// TIA Portal V19 export
FUNCTION_BLOCK "TYPIC_C501_SF_DME"   // FB55, FBD
TITLE = TYPIC_C501_SF_DME: Drukmeting
{ S7_Optimized_Access := 'TRUE' }
AUTHOR : OCOTECH
FAMILY : Typical
NAME : C501.813
// Logisch Object Besturing: C501.813
// 
// Het doel van deze subfunctie is om de algemene sturing en bediening vanuit 3B te voorzien van een drukmeting behorende tot de brandblusinstallatie.
// stored: MemoryReserve 10, SetENOAutomatically false
   VAR_INPUT
      CFG_SIG_HH { ExternalAccessible := 'False'; ExternalVisible := 'False'; ExternalWritable := 'False'} : Real;   // Schakeldrempel signalering te hoog
      CFG_SIG_H { ExternalAccessible := 'False'; ExternalVisible := 'False'; ExternalWritable := 'False'} : Real;   // Schakeldrempel signalering voorwaarschuwing hoog
      CFG_HYS_H { ExternalAccessible := 'False'; ExternalVisible := 'False'; ExternalWritable := 'False'} : Real;   // Hysteresis op signalering te hoog en voorwaarschuwing hoog
      CFG_ITYD_H { ExternalAccessible := 'False'; ExternalVisible := 'False'; ExternalWritable := 'False'} : Real;   // Tijdsvertraging signalering te hoog
      CFG_SIG_L { ExternalAccessible := 'False'; ExternalVisible := 'False'; ExternalWritable := 'False'} : Real;   // Schakeldrempel signalering te laag
      CFG_HYS_L { ExternalAccessible := 'False'; ExternalVisible := 'False'; ExternalWritable := 'False'} : Real;   // Hysteresis op signalering te laag
      CFG_ITYD_L { ExternalAccessible := 'False'; ExternalVisible := 'False'; ExternalWritable := 'False'} : Time;   // Tijdsvertraging signalering te laag
   END_VAR
   VAR_OUTPUT
      VAR_DME { ExternalAccessible := 'False'; ExternalVisible := 'False'; ExternalWritable := 'False'} : "C501_VAR_DME_TYPIC";   // Struct met alle variabelen van de drukmeting
   END_VAR
   VAR_IN_OUT
      STU_DME : "C501_STU_DME_TYPIC";   // Struct met alle sturingen vanuit de bovenliggende functie
      VAR_IF_DME : "C501_VAR_IF_DME_TYPIC";   // Struct met alle variabelen vanuit de interne sturing
   END_VAR
   VAR
      BED : Struct   // Bedieningen
         OBS : Struct   // Activeer of deactiveer de detectie van de stand van de deur van de hydrantkast
            X : "UDT_BED_ALG";
            KNOP { S7_SetPoint := 'True'} : Array[0..1] of "UDT_BED_KNOP";
         END_STRUCT;
      END_STRUCT;
      BED_OBS { ExternalWritable := 'False'} : "TYPIC_HF_BED_ALG_KNOP";   // Activeer of deactiveer de detectie van de stand van de deur van de hydrantkast
      SIG { ExternalWritable := 'False'} : Struct   // Signaleringen
         AA01 : Bool;   // Drukmeting niet observeerbaar
         AA02 : Bool;   // Storing algemeen
         AA03 : Bool;   // Druk te laag
         AA04 : Bool;   // Voorwaarschuwing druk hoog
         AA05 : Bool;   // Druk te hoog
         A001 : Bool;   // Beveiliging aangesproken
         A002 : Bool;   // Draadbreuk analoge meting
         A003 : Bool;   // Meetbereik overschreden
      END_STRUCT;
      VAR { ExternalWritable := 'False'} : Struct   // Variabelen
         RNO : USInt;   // Reden niet observeerbaar
         AUT : USInt;   // Beveiliging aangesproken
         MWA : USInt;   // Meetwaarde
         OBS { ExternalAccessible := 'False'; ExternalVisible := 'False'} : USInt;   // Observeerbaarheid
      END_STRUCT;
      HF_BST_OBS { ExternalAccessible := 'False'; ExternalVisible := 'False'; ExternalWritable := 'False'} : "TYPIC_HF_BST_OBS";   // Hulp functie besturing
   END_VAR
   // // BED.OBS.KNOP[0] : InDienst
   // // BED.OBS.KNOP[1] : UitDienst
BEGIN

REGION Network 1: START
END_REGION

REGION Network 2: +++ Bedieningen +++
   // Vrijgave en verwerking van de bedieningen (centrale en lokale bediening). De bedienwaardes worden daarna in de verdere deelfunctionaliteiten gebruikt.
END_REGION

REGION Network 3: Knoppen BED_OBS(Activeer of deactiveer de detectie van de stand van de deur van de hydrantkast)
   // Waardes en vrijge van de knoppen BED_OBS
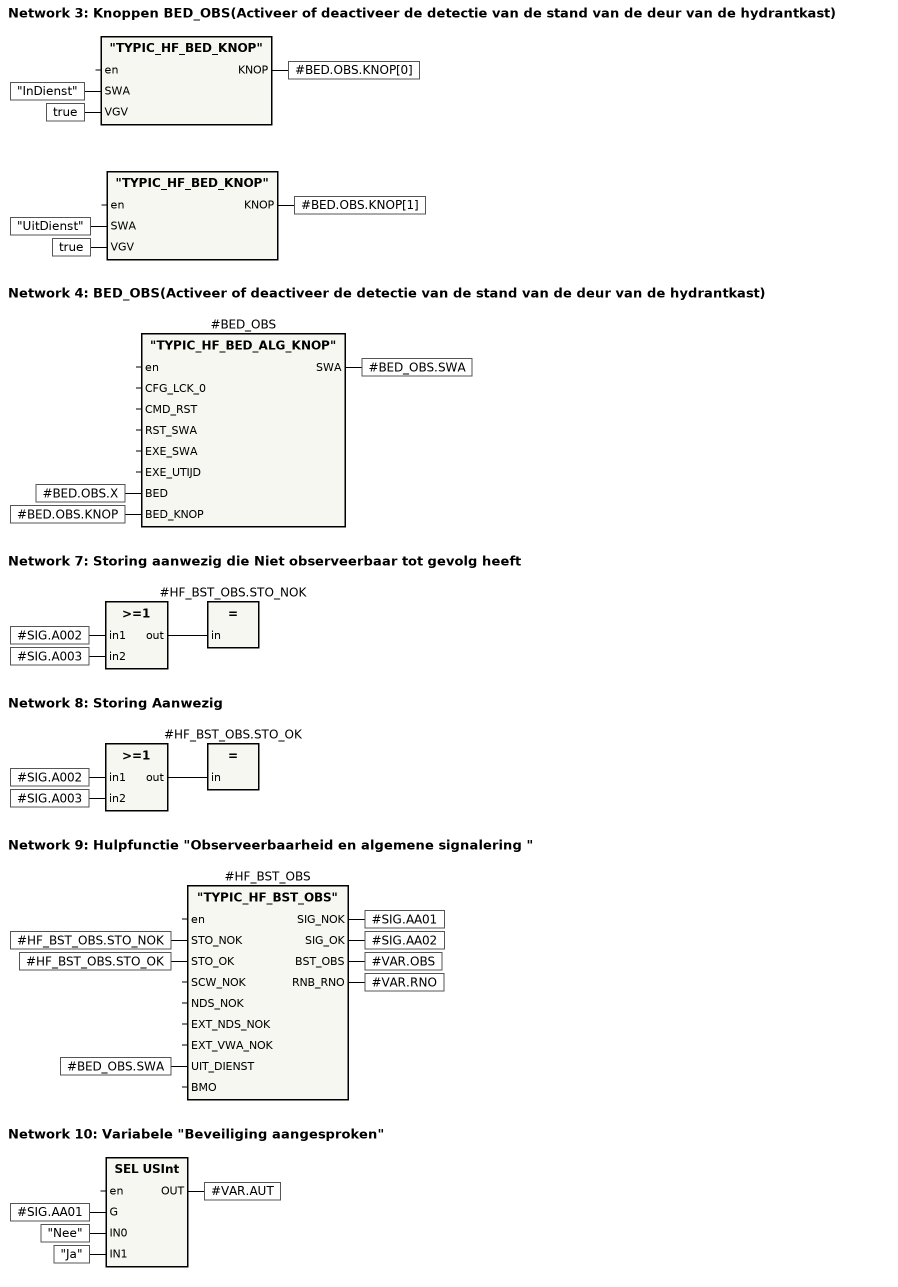
   "TYPIC_HF_BED_KNOP"(SWA := "InDienst", VGV := true, KNOP => #BED.OBS.KNOP[0]);
   "TYPIC_HF_BED_KNOP"(SWA := "UitDienst", VGV := true, KNOP => #BED.OBS.KNOP[1]);
END_REGION

REGION Network 4: BED_OBS(Activeer of deactiveer de detectie van de stand van de deur van de hydrantkast)
   // Verwerking BED_OBS
   #BED_OBS(BED := #BED.OBS.X, BED_KNOP := #BED.OBS.KNOP, SWA => #BED_OBS.SWA);   // "TYPIC_HF_BED_ALG_KNOP"
END_REGION

REGION Network 5: +++ Verwerking meetwaarde en statussen +++
   // De meetwaarde en de status wordt ontvangen vanuit de interne sturing van de drukmeting.
END_REGION

REGION Network 6: +++ Signaleringen en observeerbaarheid +++
   // Aanmaken signaleringen, bepalen observeerbaarheid (observeerbaar / niet observeerbaar) en bepalen reden niet observeerbaar.
END_REGION

REGION Network 7: Storing aanwezig die Niet observeerbaar tot gevolg heeft
   // OR-verknoping van alle storingen om input STO_BST_NOK van de hulpfunctie "Observeerbaarheid en algemene signlaring"
   #HF_BST_OBS.STO_NOK := #SIG.A002 OR #SIG.A003;
END_REGION

REGION Network 8: Storing Aanwezig
   // OR-verknoping van alle storingen om input STO_BST_OK van de hulpfunctie "Observeerbaarheid en algemene signlaring"
   #HF_BST_OBS.STO_OK := #SIG.A002 OR #SIG.A003;
END_REGION

REGION Network 9: Hulpfunctie "Observeerbaarheid en algemene signalering "
   // Bepalen variabele "Observeerbaarheid" en "reden niet Observeerbaarheid", Signaleringen "Observeerbaarheid" en "algmene storing".
   #HF_BST_OBS(STO_NOK := #HF_BST_OBS.STO_NOK,   // "TYPIC_HF_BST_OBS"
               STO_OK := #HF_BST_OBS.STO_OK,
               UIT_DIENST := #BED_OBS.SWA,
               SIG_NOK => #SIG.AA01,
               SIG_OK => #SIG.AA02,
               BST_OBS => #VAR.OBS,
               RNB_RNO => #VAR.RNO);
END_REGION

REGION Network 10: Variabele "Beveiliging aangesproken"
   // De variabele VAR_AUT geef aan of er een beveilliging aangesproken is. Deze variabele laat toe dat de verkeersoperator op SCADA kan zien of er een beveilliging aangesproken is voor deze component.
   #VAR.AUT := SEL(G := #SIG.AA01, IN0 := "Nee", IN1 := "Ja");
END_REGION

REGION Network 11 (SCL): EINDE
   // Variabelen van intern scada rakvlak naar outputs copieren
   #VAR_DME.MWA := #VAR.MWA;
   #VAR_DME.OBS := #VAR.OBS;
END_REGION
END_FUNCTION_BLOCK
